Universal Robots URScript: T009_qwen2.5-coder_32b_baseline_rep1_retry2.urscript

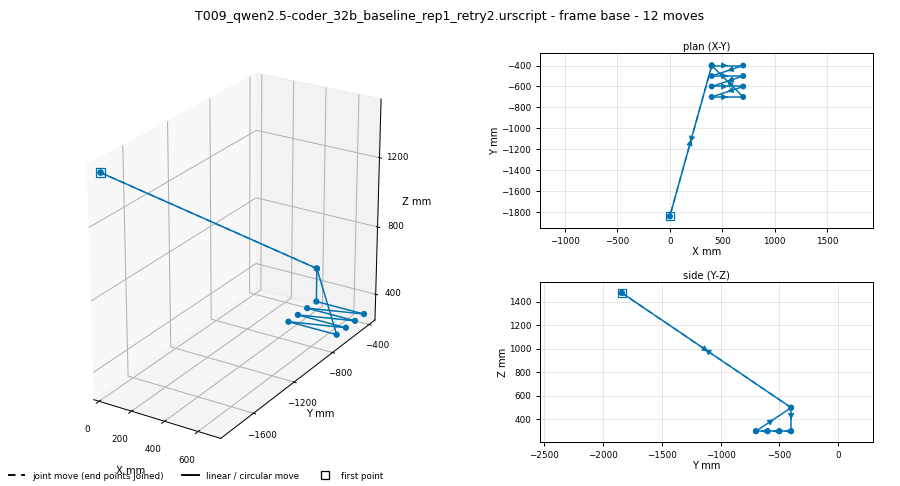
[picture p0: tool path of T009_qwen2.5-coder_32b_baseline_rep1_retry2.urscript in frame base, 12 of 12 moves have a stored position in this frame; points joined in program order, loops and branches not executed]
def laser_scan():
    # Home position
    movej(p[0.0, -1.83927, 1.47553, -1.63963, -1.14159, 0.0], a=1.2, v=1.0)

    # Above scan start
    movel(p[0.4, -0.4, 0.5, -2.2, -1.7, 0.0], a=1.2, v=0.8)

    # Descend to scan height
    movel(p[0.4, -0.4, 0.3, -2.2, -1.7, 0.0], a=1.2, v=0.5)

    # Scan line 1
    movel(p[0.7, -0.4, 0.3, -2.2, -1.7, 0.0], a=1.2, v=0.3)

    # Step to line 2
    movel(p[0.4, -0.5, 0.3, -2.2, -1.7, 0.0], a=1.2, v=0.5)

    # Scan line 2
    movel(p[0.7, -0.5, 0.3, -2.2, -1.7, 0.0], a=1.2, v=0.3)

    # Step to line 3
    movel(p[0.4, -0.6, 0.3, -2.2, -1.7, 0.0], a=1.2, v=0.5)

    # Scan line 3
    movel(p[0.7, -0.6, 0.3, -2.2, -1.7, 0.0], a=1.2, v=0.3)

    # Step to line 4
    movel(p[0.4, -0.7, 0.3, -2.2, -1.7, 0.0], a=1.2, v=0.5)

    # Scan line 4
    movel(p[0.7, -0.7, 0.3, -2.2, -1.7, 0.0], a=1.2, v=0.3)

    # Ascend from scan height
    movel(p[0.4, -0.4, 0.5, -2.2, -1.7, 0.0], a=1.2, v=0.8)

    # Return to home position
    movej(p[0.0, -1.83927, 1.47553, -1.63963, -1.14159, 0.0], a=1.2, v=1.0)

end

# Start the laser scan task
laser_scan()
